ABB RobotStudio station: RemoteControlledYumi.rspag

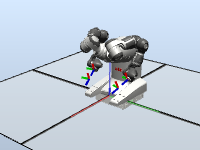
--- station ---
Station RemoteControlledYumi (saved by RobotStudio 6.5.7530.2005)
Controller IRB_14000_0.5kg_0.5m
  mechanical unit ROB_R: IRB14000_0.5_0.5_R, 6 joints, base frame (0, 0, 0) mm
  mechanical unit ROB_R_7: IRB14000_0.5_0.5_R, 1 joints, base frame (0, 0, 0) mm
  mechanical unit ROB_L: IRB14000_0.5_0.5_L, 6 joints, base frame (0, 0, 0) mm
  mechanical unit ROB_L_7: IRB14000_0.5_0.5_L, 1 joints, base frame (0, 0, 0) mm
Layout (positions relative to the parent item):
  - IRB14000_0.5_0.5 [mechanism, from Robots\IRB14000_0.5_0.5__01.rslib] at (0, 0, 0) mm
  - IRB14000_0.5_0.5_R [mechanism, from Robots\IRB14000_0.5_0.5__01.rslib] at (0, 0, 0) mm; joint values [0, -2.2689, -2.3562, 0.5236, 0, 0.6981, 0] (rad or m)
  - IRB14000_0.5_0.5_L [mechanism, from Robots\IRB14000_0.5_0.5__01.rslib] at (0, 0, 0) mm; joint values [0, -2.2689, 2.3562, 0.5236, 0, 0.6981, 0] (rad or m)
Targets, tools, work objects and paths stored in the station and not in the controller backup, written as RAPID:
! task T_ROB_R
MODULE user
  TASK PERS tooldata Servo:=[TRUE,[[0,0,114.2],[1,0,0,0]],[0.24,[8.2,12.5,48.1],[1,0,0,0],0.00022,0.00024,0.00009]];
ENDMODULE

! task T_ROB_L
MODULE user
  TASK PERS tooldata Servo:=[TRUE,[[0,0,114.2],[1,0,0,0]],[0.24,[8.2,12.5,48.1],[1,0,0,0],0.00022,0.00024,0.00009]];
ENDMODULE


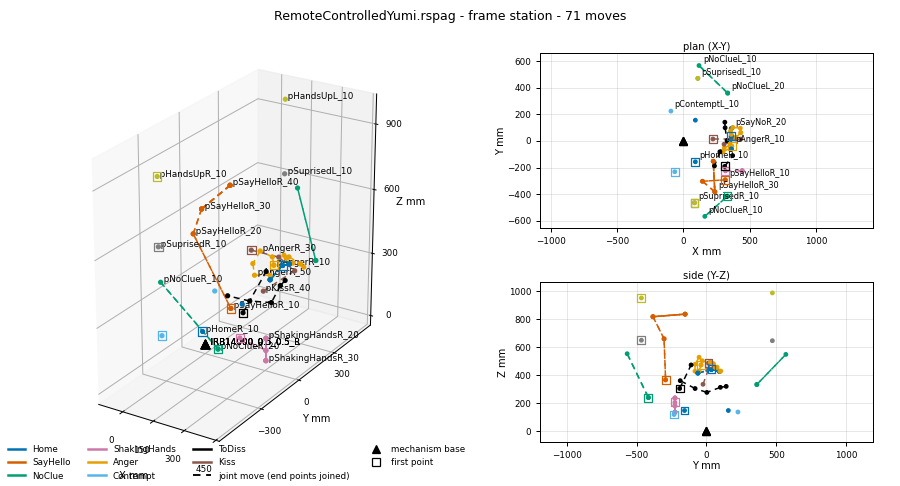
[picture p0: tool path of RemoteControlledYumi.rspag in frame station, 71 of 71 moves have a stored position in this frame; points joined in program order, loops and branches not executed]
--- Backups/IRB_14000_0.5kg_0.5m/RAPID/TASK1/PROGMOD/GesturesRight.mod ---
MODULE GesturesRight
    CONST robtarget Target_10:=[[314.699715633,-292.148031152,367.159687256],[0.159532666,0.511489136,0.162496176,0.828566947],[1,0,0,5],[-122.185137209,9E+09,9E+09,9E+09,9E+09,9E+09]];
    CONST robtarget Target_20:=[[143.244207362,-303.049195945,660.697114826],[0.6530857,-0.147210566,0.221457786,0.70905893],[1,0,0,5],[154.264930282,9E+09,9E+09,9E+09,9E+09,9E+09]];
    CONST robtarget Target_30:=[[235.909258765,-382.383017558,818.803192241],[0.490338864,0.057638645,0.190726209,0.848450999],[1,0,0,5],[-161.185793796,9E+09,9E+09,9E+09,9E+09,9E+09]];
    CONST robtarget Target_40:=[[223.935861995,-152.493872643,837.018526473],[0.280171534,-0.02496644,0.413534074,0.865950436],[1,0,0,5],[-151.318897483,9E+09,9E+09,9E+09,9E+09,9E+09]];
    CONST robtarget Target_50:=[[164.121226093,1.97602582,802.916853322],[0.202263762,-0.511536601,0.520846089,0.65279325],[0,0,0,4],[-173.792654192,9E+09,9E+09,9E+09,9E+09,9E+09]];

    CONST robtarget pKissR_10:=[[221.654761882,15.032417216,486.855961247],[0.69462356,-0.026998762,-0.017404571,0.718655868],[1,0,-2,4],[-163.076395011,9E+09,9E+09,9E+09,9E+09,9E+09]];
    CONST robtarget pKissR_20:=[[354.929073971,15.031772271,486.855510206],[0.677332175,0.151651856,0.155002452,0.702991521],[1,1,-2,4],[-128.711073694,9E+09,9E+09,9E+09,9E+09,9E+09]];
    CONST robtarget pKissR_30:=[[431.669236847,15.031318104,443.566889626],[0.639190619,0.273714512,0.272469802,0.665038289],[1,1,-2,4],[-128.711078258,9E+09,9E+09,9E+09,9E+09,9E+09]];
    CONST robtarget pKissR_40:=[[305.18930413,-24.552371649,335.517713502],[0.817106929,-0.136325958,0.414031132,0.377266114],[1,0,-2,4],[-146.11021025,9E+09,9E+09,9E+09,9E+09,9E+09]];

    CONST robtarget pSayHelloR_10:=[[314.699715633,-292.148031152,367.159687256],[0.159532666,0.511489136,0.162496176,0.828566947],[1,0,0,5],[-122.185137209,9E+09,9E+09,9E+09,9E+09,9E+09]];
    CONST robtarget pSayHelloR_20:=[[143.244207362,-303.049195945,660.697114826],[0.6530857,-0.147210566,0.221457786,0.70905893],[1,0,0,5],[154.264930282,9E+09,9E+09,9E+09,9E+09,9E+09]];
    CONST robtarget pSayHelloR_30:=[[235.909258765,-382.383017558,818.803192241],[0.490338864,0.057638645,0.190726209,0.848450999],[1,0,0,5],[-161.185793796,9E+09,9E+09,9E+09,9E+09,9E+09]];
    CONST robtarget pSayHelloR_40:=[[223.935861995,-152.493872643,837.018526473],[0.280171534,-0.02496644,0.413534074,0.865950436],[1,0,0,5],[-151.318897483,9E+09,9E+09,9E+09,9E+09,9E+09]];

    CONST robtarget pNoClueR_20:=[[331.005027183,-415.055262019,240.258080351],[0.395586627,0.754614135,0.446136315,0.273918084],[0,0,0,5],[-121.777862862,9E+09,9E+09,9E+09,9E+09,9E+09]];
    CONST robtarget pNoClueR_10:=[[160.547655799,-566.897146043,554.058433096],[0.765286197,0.45290272,-0.146899327,0.433170579],[1,0,0,5],[169.961367293,9E+09,9E+09,9E+09,9E+09,9E+09]];

    CONST robtarget pHomeR_10:=[[89.387946422,-156.622117956,147.913470217],[0.066010726,-0.842420918,-0.111214912,-0.523068661],[0,0,0,4],[-101.964427132,9E+09,9E+09,9E+09,9E+09,9E+09]];

    CONST robtarget pShakingHandsR_10:=[[315.738569474,-225.378667241,206.19666017],[0.339537865,-0.658753284,0.219946518,-0.63433562],[0,0,1,4],[-108.735165241,9E+09,9E+09,9E+09,9E+09,9E+09]];
    CONST robtarget pShakingHandsR_40:=[[440.955889424,-225.380066174,182.362206426],[0.11092253,0.699479671,0.098185544,0.699130876],[1,1,-1,4],[-108.735179691,9E+09,9E+09,9E+09,9E+09,9E+09]];
    CONST robtarget pShakingHandsR_20:=[[440.955617046,-225.379654836,237.561937878],[0.110922498,0.699479548,0.098185209,0.699131051],[1,2,-1,4],[-108.735186134,9E+09,9E+09,9E+09,9E+09,9E+09]];
    CONST robtarget pShakingHandsR_30:=[[440.955691509,-225.379895287,135.696714265],[0.110922513,0.699479626,0.098185285,0.69913096],[1,1,-1,4],[-108.735178424,9E+09,9E+09,9E+09,9E+09,9E+09]];

    CONST robtarget pAngerR_10:=[[363.531838424,-38.636637831,473.352200394],[0.300745531,-0.136482013,-0.04783233,-0.94267537],[1,0,0,4],[-130.403991592,9E+09,9E+09,9E+09,9E+09,9E+09]];
    CONST robtarget pAngerR_20:=[[350.75125662,-29.515051373,503.763471562],[0.257706669,0.015454476,-0.043694396,-0.965110995],[1,0,0,4],[-121.508331805,9E+09,9E+09,9E+09,9E+09,9E+09]];
    CONST robtarget pAngerR_30:=[[306.632986283,-52.601439571,528.928808016],[0.261410738,0.064341961,-0.04557113,-0.96200198],[1,0,0,4],[-122.099256333,9E+09,9E+09,9E+09,9E+09,9E+09]];
    CONST robtarget pAngerR_40:=[[288.800844629,-81.29752225,478.773158089],[0.216079199,-0.014900154,-0.132940712,-0.967168306],[1,0,0,4],[-129.63023687,9E+09,9E+09,9E+09,9E+09,9E+09]];
    CONST robtarget pAngerR_50:=[[297.418539835,-81.958124122,428.713986694],[0.109438137,-0.189120514,-0.255285462,-0.941852461],[1,0,0,4],[-136.020526211,9E+09,9E+09,9E+09,9E+09,9E+09]];
    CONST robtarget pAngerR_60:=[[354.350248531,-52.04234992,430.466884854],[0.177313873,-0.133250362,-0.160013373,-0.961873096],[1,0,0,4],[-129.960312977,9E+09,9E+09,9E+09,9E+09,9E+09]];

    CONST robtarget pContemptR_10:=[[-65.408295514,-231.499226874,119.303275828],[0.188476781,-0.180789855,-0.941418807,0.213359232],[1,0,-1,5],[-169.723005722,9E+09,9E+09,9E+09,9E+09,9E+09]];

    CONST robtarget pToDissR_10:=[[310.08261334,-191.393706007,305.466074161],[0.673664037,0.094173277,0.328608316,0.655228765],[1,0,-1,4],[-103.279379297,9E+09,9E+09,9E+09,9E+09,9E+09]];
    CONST robtarget pToDissR_20:=[[370.062778661,-109.65260016,473.851053749],[0.666629844,-0.160646787,-0.045141606,0.726470575],[1,0,-1,4],[-103.911686462,9E+09,9E+09,9E+09,9E+09,9E+09]];

    CONST robtarget pSuprisedR_10:=[[83.03148877,-465.085929834,650.386646622],[0.703838382,-0.01527703,0.013249227,-0.710072252],[1,0,-2,4],[115.639447021,9E+09,9E+09,9E+09,9E+09,9E+09]];

    CONST robtarget pHandsUpR_10:=[[83.03187344,-465.085940939,952.690090127],[0.703838421,-0.015277226,0.013249253,-0.710072208],[0,1,-2,4],[137.877026865,9E+09,9E+09,9E+09,9E+09,9E+09]];

    CONST robtarget pSayNoR_10:=[[359.801557873,36.119395579,442.32851368],[0.724497161,0.007725768,-0.00165855,-0.68923249],[1,0,0,4],[-143.857840595,9E+09,9E+09,9E+09,9E+09,9E+09]];
    CONST robtarget pSayNoR_20:=[[359.802142459,93.128614528,426.773071438],[0.708401181,-0.152065476,-0.153449882,-0.671935259],[1,0,0,4],[-143.857842721,9E+09,9E+09,9E+09,9E+09,9E+09]];
    CONST robtarget pSayNoR_30:=[[359.802673586,-61.261892837,415.421024536],[0.687551152,0.228536622,0.208835913,-0.656834824],[1,0,0,4],[-143.857842589,9E+09,9E+09,9E+09,9E+09,9E+09]];

    VAR syncident syncToDiss;

    PROC Home()
        MoveJ pHomeR_10,v1000,fine,Servo\WObj:=wobj0;
    ENDPROC

    PROC SayHello()
        MoveJ pSayHelloR_10,v1000,z10,Servo\WObj:=wobj0;
        MoveJ pSayHelloR_20,v1000,z10,Servo\WObj:=wobj0;
        MoveJ pSayHelloR_30,v400,z10,Servo\WObj:=wobj0;
        MoveJ pSayHelloR_40,v400,z10,Servo\WObj:=wobj0;
        MoveJ pSayHelloR_30,v400,z10,Servo\WObj:=wobj0;
        MoveJ pSayHelloR_40,v400,z10,Servo\WObj:=wobj0;
        MoveJ pSayHelloR_40,v400,z10,Servo\WObj:=wobj0;
        MoveJ pSayHelloR_30,v400,z10,Servo\WObj:=wobj0;
        MoveJ pSayHelloR_20,v1000,z10,Servo\WObj:=wobj0;
        MoveJ pSayHelloR_10,v1000,z10,Servo\WObj:=wobj0;
        Home;
    ENDPROC

    PROC NoClue()
        MoveJ pNoClueR_20,v1000,z10,Servo\WObj:=wobj0;
        MoveJ pNoClueR_10,v1000,z10,Servo\WObj:=wobj0;
        WaitTime 2;
        MoveJ pNoClueR_20,v1000,z10,Servo\WObj:=wobj0;
        Home;
    ENDPROC

    PROC ShakingHands()
        MoveJ pShakingHandsR_10,v1000,z10,Servo\WObj:=wobj0;
        MoveJ pShakingHandsR_40,v1000,z10,Servo\WObj:=wobj0;
        WaitTime 1;
        MoveJ pShakingHandsR_20,v1000,z10,Servo\WObj:=wobj0;
        MoveJ pShakingHandsR_30,v1000,z10,Servo\WObj:=wobj0;
        MoveJ pShakingHandsR_20,v1000,z10,Servo\WObj:=wobj0;
        MoveJ pShakingHandsR_30,v1000,z10,Servo\WObj:=wobj0;
        MoveJ pShakingHandsR_20,v1000,z10,Servo\WObj:=wobj0;
        MoveJ pShakingHandsR_30,v1000,z10,Servo\WObj:=wobj0;
        MoveJ pShakingHandsR_40,v1000,z10,Servo\WObj:=wobj0;
        WaitTime 1;
        Home;
    ENDPROC

    PROC Anger()
        MoveJ pAngerR_10,v1000,z40,Servo\WObj:=wobj0;
        MoveJ pAngerR_20,v1000,z40,Servo\WObj:=wobj0;
        MoveJ pAngerR_30,v1000,z40,Servo\WObj:=wobj0;
        MoveJ pAngerR_40,v1000,z40,Servo\WObj:=wobj0;
        MoveJ pAngerR_50,v1000,z40,Servo\WObj:=wobj0;
        MoveJ pAngerR_60,v1000,z40,Servo\WObj:=wobj0;
        MoveJ pAngerR_10,v1000,z40,Servo\WObj:=wobj0;
        Home;
    ENDPROC

    PROC Contempt()
        MoveJ pContemptR_10,v1000,z10,Servo\WObj:=wobj0;
        WaitTime 2;
        Home;
    ENDPROC

    PROC ToDiss()
        MoveJ pToDissR_10,v500,z10,Servo\WObj:=wobj0;
        MoveJ pToDissR_20,v500,z10,Servo\WObj:=wobj0;
        !Restore sync
        !WaitSyncTask syncToDiss, task_list;
        WaitTime 1;
        Home;
    ENDPROC

    PROC Kiss()
        MoveJ pKissR_10,v1000,z10,Servo\WObj:=wobj0;
        MoveJ pKissR_20,v1000,z10,Servo\WObj:=wobj0;
        MoveJ pKissR_30,v1000,z10,Servo\WObj:=wobj0;
        MoveJ pKissR_40,v1000,z10,Servo\WObj:=wobj0;
        Home;
    ENDPROC

    PROC Suprised()
        MoveJ pSuprisedR_10,v5000,z10,Servo\WObj:=wobj0;
        WaitTime 2;
        Home;
    ENDPROC

    PROC HandsUp()
        MoveJ pHandsUpR_10,v1000,z10,Servo\WObj:=wobj0;
        WaitTime 2;
        Home;
    ENDPROC

    PROC SayNo()
        MoveJ pSayNoR_10,v1000,z10,Servo\WObj:=wobj0;
        MoveJ pSayNoR_20,v1000,z10,Servo\WObj:=wobj0;
        MoveJ pSayNoR_10,v1000,z10,Servo\WObj:=wobj0;
        MoveJ pSayNoR_30,v1000,z10,Servo\WObj:=wobj0;
        MoveJ pSayNoR_10,v1000,z10,Servo\WObj:=wobj0;
        MoveJ pSayNoR_20,v1000,z10,Servo\WObj:=wobj0;
        MoveJ pSayNoR_10,v1000,z10,Servo\WObj:=wobj0;
        MoveJ pSayNoR_30,v1000,z10,Servo\WObj:=wobj0;
        MoveJ pSayNoR_10,v1000,z10,Servo\WObj:=wobj0;
        MoveJ pSayNoR_20,v1000,z10,Servo\WObj:=wobj0;
        MoveJ pSayNoR_10,v1000,z10,Servo\WObj:=wobj0;
        MoveJ pSayNoR_30,v1000,z10,Servo\WObj:=wobj0;
        MoveJ pSayNoR_10,v1000,z10,Servo\WObj:=wobj0;
        Home;
    ENDPROC

ENDMODULE

--- Backups/IRB_14000_0.5kg_0.5m/RAPID/TASK1/PROGMOD/MainModule.mod ---
MODULE MainModule
    ! This procedure is the entry point when starting a simulation.
    PROC main()
        Init;
        RunLoop;
    ENDPROC
ENDMODULE

--- Backups/IRB_14000_0.5kg_0.5m/RAPID/TASK1/PROGMOD/Remote.mod ---
MODULE Remote
    TASK PERS bool bStart:=FALSE;
    TASK PERS bool bRunning:=FALSE;

    TASK PERS string stName:="NoClue";

    PROC Init()
        bStart:=FALSE;
        bRunning:=FALSE;
    ENDPROC

    PROC RunLoop()
        Init;
        WHILE TRUE DO
            WaitUntil bStart;
            bRunning:=TRUE;
            bStart:=FALSE;
            %stName %;
            bRunning:=FALSE;
        ENDWHILE
    ENDPROC
ENDMODULE

--- Backups/IRB_14000_0.5kg_0.5m/RAPID/TASK1/SYSMOD/LINKEDM.sys ---
%%%
  VERSION:1
  LANGUAGE:ENGLISH
%%%

MODULE LINKEDM (SYSMODULE)

! FOLLOWER
!     Name of electronically linked follower axis used by operator at teach pendent.
      PERS string l_f_axis_name{5}       :=  ["",  "", "", "", ""];

!     Name of the mechanical unit for follower axis.
      PERS string l_f_mecunt_n{5}  :=  ["", "", "", "", ""];

!     Linked follower axis number in the mechanical unit (first axis in mech. unit is number 1).
      PERS num l_f_axis_no{5}      :=  [0,          0,   0,  0,  0];

! MASTER
!     Name of the mechanical unit for linked master axis.
      PERS string l_m_mecunt_n{5} :=  ["", "", "", "", ""];

!     Linked master axis number in the mechanical unit (first axis in mech. unit is number 1).
!     See axis number table in documentation for different master mechanical units.
      PERS num l_m_axis_no{5}     :=  [0,  0,  0,  0,  0];

! POSITION OFFSET
!     The increase of the allowed offset position between the master and follower
!     positions, used when starting AUTO mode. As soon as the offset is decreased
!     the old configurated parameter is used.
!     Example: 3 => the configurated value of allowed offset is increased 3 times.
      PERS num offset_ratio{5}       :=  [10,  10,   10,  10,  10];

! SPEED RATIO
!     Speed_ratio used in AUTO and JOG modes [ very_slow   slow    normal    fast]
!     Value 1 = max allowed manual speed.
      CONST num speed_ratio {20}      := [0.01, 0.01, 0.01, 0.01, 0.01,
                                          0.05, 0.05, 0.05, 0.05, 0.05,
                                          0.20, 0.20, 0.20, 0.20, 0.20,
                                          1.00, 1.00, 1.00, 1.00, 1.00];

! STEP SIZE
!     Displacement position used in JOG mode for each activation of positive or
!     negative movement.                  [very_short    short   normal   long]
!     Unit degees or meter.
      CONST num displacement {20}     := [0.001, 0.001, 0.001, 0.001, 0.001,
                                          0.005, 0.005, 0.005, 0.005, 0.005,
                                          0.020, 0.020, 0.020, 0.020, 0.020,
                                          0.100, 0.100, 0.100, 0.100, 0.100];


!-------------------------------------------------------------
 PROC Linked_m ()
      Linked_m_exe ;
 ENDPROC
ENDMODULE

--- Backups/IRB_14000_0.5kg_0.5m/RAPID/TASK2/PROGMOD/GesturesLeft.mod ---
MODULE GesturesLeft
    CONST robtarget pContemptL_10:=[[-94.491553607,225.077568886,137.327093089],[0.306193092,0.231227469,-0.892125882,-0.238518467],[-1,0,1,5],[170.068678796,9E+09,9E+09,9E+09,9E+09,9E+09]];

    CONST robtarget pAngerL_10:=[[431.098301309,61.959159256,458.125646738],[0.188343319,-0.135994051,0.205422096,-0.950701938],[-1,0,1,4],[116.357977607,9E+09,9E+09,9E+09,9E+09,9E+09]];
    CONST robtarget pAngerL_20:=[[427.541303481,96.078854268,428.274281879],[0.242851724,-0.180947804,0.292829472,-0.906935407],[-1,0,1,4],[121.814803059,9E+09,9E+09,9E+09,9E+09,9E+09]];
    CONST robtarget pAngerL_30:=[[371.370802791,102.647922136,430.309317662],[0.250175091,-0.189729403,0.368594998,-0.874958802],[-1,0,1,4],[129.017692817,9E+09,9E+09,9E+09,9E+09,9E+09]];
    CONST robtarget pAngerL_40:=[[354.020430947,75.987991242,458.212372351],[0.211781199,-0.1200539,0.309854599,-0.919089719],[-1,0,1,4],[127.31237471,9E+09,9E+09,9E+09,9E+09,9E+09]];
    CONST robtarget pAngerL_50:=[[359.09325296,50.040718323,483.103930387],[0.132670971,-0.022575789,0.326351779,-0.935619187],[-1,0,1,4],[134.887718951,9E+09,9E+09,9E+09,9E+09,9E+09]];
    CONST robtarget pAngerL_60:=[[396.062972248,27.911166703,492.703033028],[0.114272503,-0.022558134,0.275782172,-0.954136845],[-1,0,1,4],[129.639362388,9E+09,9E+09,9E+09,9E+09,9E+09]];

    CONST robtarget pToDissL_10:=[[311.262788205,141.365155063,320.620976131],[0.30127594,0.413850338,-0.12183377,0.850363004],[-1,0,0,4],[109.137922493,9E+09,9E+09,9E+09,9E+09,9E+09]];
    CONST robtarget pToDissL_20:=[[313.163869898,99.550091581,313.678214603],[0.405584331,0.369718383,-0.180052484,0.816327612],[-1,0,0,4],[120.550323233,9E+09,9E+09,9E+09,9E+09,9E+09]];
    CONST robtarget pToDissL_30:=[[327.793203037,3.134311337,277.462215839],[0.525517576,0.35593926,-0.443885036,0.632538216],[-1,0,0,4],[161.707001678,9E+09,9E+09,9E+09,9E+09,9E+09]];
    CONST robtarget pToDissL_40:=[[274.023321791,-80.991562457,305.086937965],[0.647848865,0.227051384,-0.451204352,0.570222895],[-1,0,0,4],[171.12747593,9E+09,9E+09,9E+09,9E+09,9E+09]];
    CONST robtarget pToDissL_50:=[[233.086731165,-187.421735572,361.300083015],[0.647848463,0.227050931,-0.451204503,0.570223413],[-1,1,-1,4],[154.498524311,9E+09,9E+09,9E+09,9E+09,9E+09]];

    CONST robtarget pHomeL_10:=[[89.387946423,156.622117957,147.913470217],[0.066010726,0.842420918,-0.111214912,0.523068661],[0,0,0,4],[101.964427132,9E+09,9E+09,9E+09,9E+09,9E+09]];

    CONST robtarget pSuprisedL_10:=[[108.153191894,471.411528047,647.230762026],[0.699371757,0.003098078,0.006552088,-0.714721357],[-1,0,0,4],[-132.382826108,9E+09,9E+09,9E+09,9E+09,9E+09]];

    CONST robtarget pHandsUpL_10:=[[108.153567372,471.411547841,988.720364525],[0.699371728,0.003098049,0.006552252,-0.714721384],[0,-1,0,4],[-132.382818416,9E+09,9E+09,9E+09,9E+09,9E+09]];

    CONST robtarget pNoClueL_10:=[[116.844170561,567.745373907,549.176802943],[0.612414859,-0.27944775,-0.40047322,-0.621673705],[-1,0,0,5],[170.97345488,9E+09,9E+09,9E+09,9E+09,9E+09]];
    CONST robtarget pNoClueL_20:=[[332.599072052,360.424339744,333.84998915],[0.323491568,-0.733582932,-0.040436016,-0.596300441],[-1,0,0,5],[100.391786771,9E+09,9E+09,9E+09,9E+09,9E+09]];

    VAR syncident syncToDiss;

    PROC Home()
        MoveJ pHomeL_10,v1000,fine,Servo\WObj:=wobj0;
    ENDPROC

    PROC Anger()
        MoveJ pAngerL_10,v1000,z40,Servo\WObj:=wobj0;
        MoveJ pAngerL_20,v1000,z40,Servo\WObj:=wobj0;
        MoveJ pAngerL_30,v1000,z40,Servo\WObj:=wobj0;
        MoveJ pAngerL_40,v1000,z40,Servo\WObj:=wobj0;
        MoveJ pAngerL_50,v1000,z40,Servo\WObj:=wobj0;
        MoveJ pAngerL_60,v1000,z40,Servo\WObj:=wobj0;
        MoveJ pAngerL_10,v1000,z40,Servo\WObj:=wobj0;
        Home;
    ENDPROC

    PROC Contempt()
        MoveJ pContemptL_10,v1000,z10,Servo\WObj:=wobj0;
        WaitTime 2;
        Home;
    ENDPROC

    PROC ToDiss()
        MoveJ pToDissL_10,v1000,z10,Servo\WObj:=wobj0;
        MoveJ pToDissL_20,v1000,z10,Servo\WObj:=wobj0;
        MoveJ pToDissL_30,v1000,z10,Servo\WObj:=wobj0;
        MoveJ pToDissL_40,v1000,z10,Servo\WObj:=wobj0;
        MoveJ pToDissL_50,v1000,fine,Servo\WObj:=wobj0;
        ! Restore sync
        ! WaitSyncTask syncToDiss, task_list;
        WaitTime 1;
        Home;
    ENDPROC

    PROC Suprised()
        MoveJ pSuprisedL_10,v5000,z10,Servo\WObj:=wobj0;
        WaitTime 2;
        Home;
    ENDPROC

    PROC HandsUp()
        MoveJ pHandsUpL_10,v1000,z10,Servo\WObj:=wobj0;
        WaitTime 2;
        Home;
    ENDPROC

    PROC NoClue()
        MoveJ pNoClueL_20,v1000,z10,Servo\WObj:=wobj0;
        MoveJ pNoClueL_10,v1000,z10,Servo\WObj:=wobj0;
        WaitTime 2;
        MoveJ pNoClueL_20,v1000,z10,Servo\WObj:=wobj0;
        Home;
    ENDPROC
ENDMODULE

--- Backups/IRB_14000_0.5kg_0.5m/SYSPAR/EIO.cfg ---
EIO:CFG_1.0:6:1::
#
SYSSIG_IN:

      -Signal "Collision_Avoidance" -Action "CollAvoidance"
#
INDUSTRIAL_NETWORK:

      -Name "EtherNetIP" -Connection "Private Network"\
      -Label "EtherNet/IP Adapter Network"

      -Name "DeviceNet" -Label "DeviceNet Master/Slave Network" -Address "2"
#
EIO_CROSS:

      -Name "Cross_Signal_Lamp" -Res "Signal_Lamp" -Act1 "DRV1BRAKE"
#
EIO_SIGNAL_SAFELEVEL:

      -Name "FlangePowerSafeLevel" -ActionWhenStartup "Last"
#
DEVICENET_DEVICE:

      -Name "D652_10" -VendorName "ABB Robotics" -ProductName "24 VDC Unit"\
      -Address 10 -ProductCode 26 -DeviceType 7 -ConnectionType "COS"\
      -OutputSize 2 -InputSize 2
#
DEVICENET_INTERNAL_DEVICE:

      -Name "DN_Internal_Device" -VendorName "ABB Robotics"\
      -ProductName "DeviceNet Internal Slave Device"
#
ETHERNETIP_INTERNAL_DEVICE:

      -Name "EN_Internal_Device" -VendorName "ABB Robotics"\
      -ProductName "EtherNet/IP Internal Adapter Device"
#
EIO_SIGNAL:

      -Name "custom_DI_0" -SignalType "DI" -Device "D652_10" -DeviceMap "0"

      -Name "custom_DI_1" -SignalType "DI" -Device "D652_10" -DeviceMap "1"

      -Name "custom_DI_2" -SignalType "DI" -Device "D652_10" -DeviceMap "2"

      -Name "custom_DI_3" -SignalType "DI" -Device "D652_10" -DeviceMap "3"

      -Name "custom_DI_4" -SignalType "DI" -Device "D652_10" -DeviceMap "4"

      -Name "custom_DI_5" -SignalType "DI" -Device "D652_10" -DeviceMap "5"

      -Name "custom_DI_6" -SignalType "DI" -Device "D652_10" -DeviceMap "6"

      -Name "custom_DI_7" -SignalType "DI" -Device "D652_10" -DeviceMap "7"

      -Name "custom_DO_0" -SignalType "DO" -Device "D652_10" -DeviceMap "0"

      -Name "custom_DO_1" -SignalType "DO" -Device "D652_10" -DeviceMap "1"

      -Name "custom_DO_2" -SignalType "DO" -Device "D652_10" -DeviceMap "2"

      -Name "custom_DO_3" -SignalType "DO" -Device "D652_10" -DeviceMap "3"

      -Name "custom_DO_4" -SignalType "DO" -Device "D652_10" -DeviceMap "4"

      -Name "custom_DO_5" -SignalType "DO" -Device "D652_10" -DeviceMap "5"

      -Name "custom_DO_6" -SignalType "DO" -Device "D652_10" -DeviceMap "6"

      -Name "custom_DO_7" -SignalType "DO" -Device "D652_10" -DeviceMap "7"

      -Name "hall_sensor_joint_1" -SignalType "DI" -Device "D652_10"\
      -DeviceMap "8"

      -Name "hall_sensor_joint_2" -SignalType "DI" -Device "D652_10"\
      -DeviceMap "9"

      -Name "hall_sensor_joint_3" -SignalType "DI" -Device "D652_10"\
      -DeviceMap "11"

      -Name "hall_sensor_joint_4" -SignalType "DI" -Device "D652_10"\
      -DeviceMap "12"

      -Name "hall_sensor_joint_5" -SignalType "DI" -Device "D652_10"\
      -DeviceMap "13"

      -Name "hall_sensor_joint_6" -SignalType "DI" -Device "D652_10"\
      -DeviceMap "14"

      -Name "hall_sensor_joint_7" -SignalType "DI" -Device "D652_10"\
      -DeviceMap "10"

      -Name "hall_sensor_24V_ROB_R" -SignalType "DO" -Device "D652_10"\
      -DeviceMap "8"

      -Name "hall_sensor_24V_ROB_L" -SignalType "DO" -Device "D652_10"\
      -DeviceMap "9"

      -Name "flange_24V_ROB_R" -SignalType "DO" -Device "D652_10"\
      -DeviceMap "10" -SafeLevel "FlangePowerSafeLevel"

      -Name "flange_24V_ROB_L" -SignalType "DO" -Device "D652_10"\
      -DeviceMap "11" -SafeLevel "FlangePowerSafeLevel"

      -Name "Signal_Lamp" -SignalType "DO" -Device "D652_10" -DeviceMap "12"

      -Name "Collision_Avoidance" -SignalType "DO" -Access "All" -Default 1
